// TIA Portal V19 export
TYPE "LEXCHANGETRAY_typeConstraintRollerEm_xPositionAxis_monitor"
// stored: Access Published
   STRUCT
      posIndex : Int;
   END_STRUCT;
END_TYPE
